FUNCTION_BLOCK Feedforward (* Composite Function Block Type *)
  (* Standard: 61499-2 *)
  (* Version 0.0, 2018-09-24, 4DIAC-IDE, 4DIAC-Consortium *)
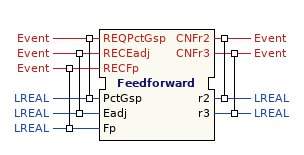
  EVENT_INPUT
    REQPctGsp WITH PctGsp;
    RECEadj WITH Eadj;
    RECFp WITH Fp;
  END_EVENT
  EVENT_OUTPUT
    CNFr2 WITH r2;
    CNFr3 WITH r3;
  END_EVENT
  VAR_INPUT
    PctGsp : LREAL;
    Eadj : LREAL;
    Fp : LREAL;
  END_VAR
  VAR_OUTPUT
    r2 : LREAL;
    r3 : LREAL;
  END_VAR
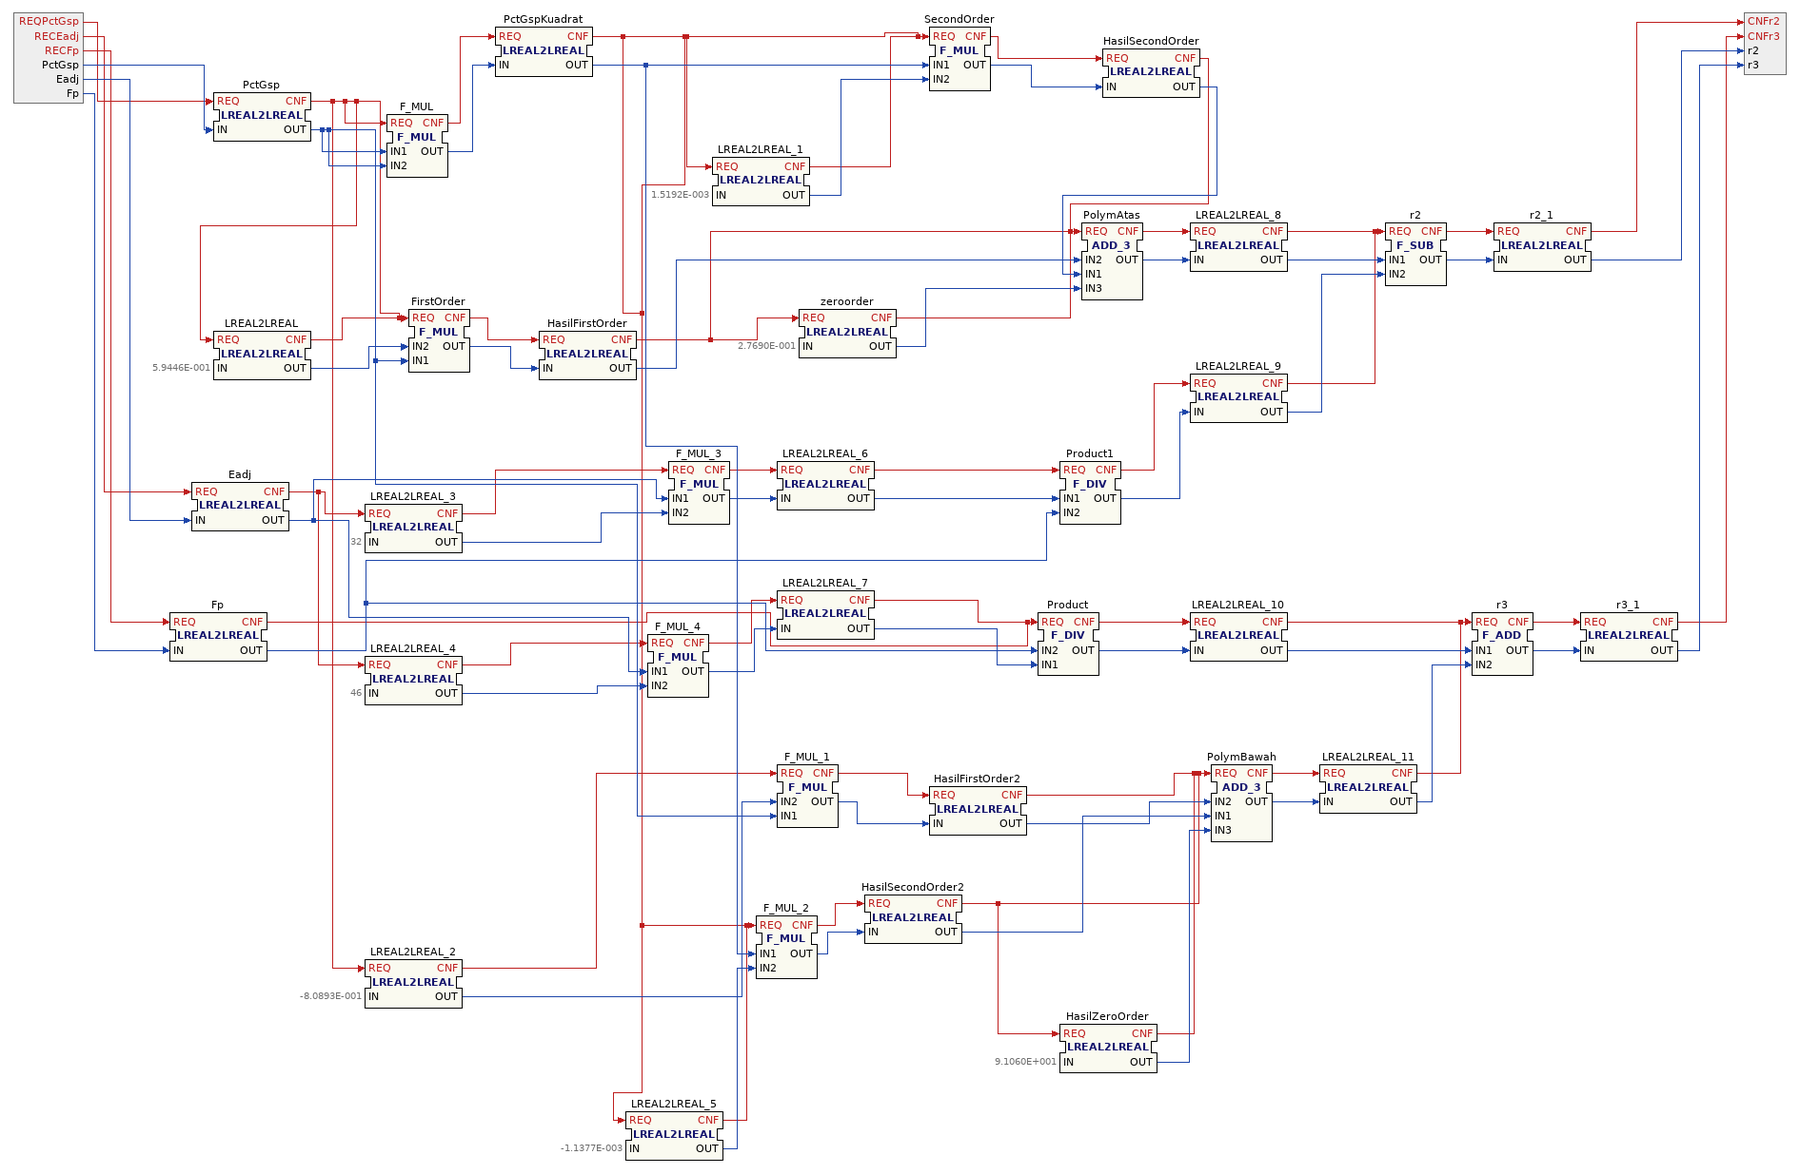
  FBS
    PctGsp : LREAL2LREAL;
    Eadj : LREAL2LREAL;
    Fp : LREAL2LREAL;
    F_MUL : F_MUL;
    PctGspKuadrat : LREAL2LREAL;
    LREAL2LREAL : LREAL2LREAL(IN := 5.9446E-001);
    LREAL2LREAL_1 : LREAL2LREAL(IN := 1.5192E-003);
    HasilFirstOrder : LREAL2LREAL;
    HasilSecondOrder : LREAL2LREAL;
    zeroorder : LREAL2LREAL(IN := 2.7690E-001);
    FirstOrder : F_MUL;
    PolymAtas : ADD_3;
    SecondOrder : F_MUL;
    PolymBawah : ADD_3;
    LREAL2LREAL_2 : LREAL2LREAL(IN := -8.0893E-001);
    F_MUL_1 : F_MUL;
    HasilFirstOrder2 : LREAL2LREAL;
    HasilSecondOrder2 : LREAL2LREAL;
    LREAL2LREAL_5 : LREAL2LREAL(IN := -1.1377E-003);
    F_MUL_2 : F_MUL;
    HasilZeroOrder : LREAL2LREAL(IN := 9.1060E+001);
    LREAL2LREAL_3 : LREAL2LREAL(IN := 32);
    LREAL2LREAL_4 : LREAL2LREAL(IN := 46);
    F_MUL_3 : F_MUL;
    F_MUL_4 : F_MUL;
    LREAL2LREAL_6 : LREAL2LREAL;
    LREAL2LREAL_7 : LREAL2LREAL;
    Product1 : F_DIV;
    Product : F_DIV;
    r2 : F_SUB;
    LREAL2LREAL_8 : LREAL2LREAL;
    LREAL2LREAL_9 : LREAL2LREAL;
    LREAL2LREAL_10 : LREAL2LREAL;
    r3 : F_ADD;
    LREAL2LREAL_11 : LREAL2LREAL;
    r2_1 : LREAL2LREAL;
    r3_1 : LREAL2LREAL;
  END_FBS
  EVENT_CONNECTIONS
    REQPctGsp TO PctGsp.REQ;
    RECEadj TO Eadj.REQ;
    RECFp TO Fp.REQ;
    PctGsp.CNF TO F_MUL.REQ;
    F_MUL.CNF TO PctGspKuadrat.REQ;
    PctGsp.CNF TO LREAL2LREAL.REQ;
    LREAL2LREAL.CNF TO FirstOrder.REQ;
    PctGsp.CNF TO FirstOrder.REQ;
    FirstOrder.CNF TO HasilFirstOrder.REQ;
    HasilFirstOrder.CNF TO PolymAtas.REQ;
    LREAL2LREAL_1.CNF TO SecondOrder.REQ;
    PctGspKuadrat.CNF TO SecondOrder.REQ;
    PctGspKuadrat.CNF TO LREAL2LREAL_1.REQ;
    SecondOrder.CNF TO HasilSecondOrder.REQ;
    HasilSecondOrder.CNF TO PolymAtas.REQ;
    zeroorder.CNF TO PolymAtas.REQ;
    HasilFirstOrder.CNF TO zeroorder.REQ;
    PctGsp.CNF TO LREAL2LREAL_2.REQ;
    LREAL2LREAL_2.CNF TO F_MUL_1.REQ;
    F_MUL_1.CNF TO HasilFirstOrder2.REQ;
    HasilFirstOrder2.CNF TO PolymBawah.REQ;
    HasilSecondOrder2.CNF TO PolymBawah.REQ;
    F_MUL_2.CNF TO HasilSecondOrder2.REQ;
    PctGspKuadrat.CNF TO F_MUL_2.REQ;
    LREAL2LREAL_5.CNF TO F_MUL_2.REQ;
    PctGspKuadrat.CNF TO LREAL2LREAL_5.REQ;
    HasilZeroOrder.CNF TO PolymBawah.REQ;
    HasilSecondOrder2.CNF TO HasilZeroOrder.REQ;
    Eadj.CNF TO LREAL2LREAL_4.REQ;
    Eadj.CNF TO LREAL2LREAL_3.REQ;
    LREAL2LREAL_4.CNF TO F_MUL_4.REQ;
    LREAL2LREAL_3.CNF TO F_MUL_3.REQ;
    F_MUL_3.CNF TO LREAL2LREAL_6.REQ;
    LREAL2LREAL_6.CNF TO Product1.REQ;
    F_MUL_4.CNF TO LREAL2LREAL_7.REQ;
    LREAL2LREAL_7.CNF TO Product.REQ;
    Fp.CNF TO Product.REQ;
    PolymAtas.CNF TO LREAL2LREAL_8.REQ;
    LREAL2LREAL_8.CNF TO r2.REQ;
    LREAL2LREAL_9.CNF TO r2.REQ;
    Product1.CNF TO LREAL2LREAL_9.REQ;
    Product.CNF TO LREAL2LREAL_10.REQ;
    LREAL2LREAL_10.CNF TO r3.REQ;
    PolymBawah.CNF TO LREAL2LREAL_11.REQ;
    LREAL2LREAL_11.CNF TO r3.REQ;
    r2_1.CNF TO CNFr2;
    r2.CNF TO r2_1.REQ;
    r3.CNF TO r3_1.REQ;
    r3_1.CNF TO CNFr3;
  END_CONNECTIONS
  DATA_CONNECTIONS
    Fp TO Fp.IN;
    PctGsp TO PctGsp.IN;
    PctGsp.OUT TO F_MUL.IN1;
    PctGsp.OUT TO F_MUL.IN2;
    F_MUL.OUT TO PctGspKuadrat.IN;
    LREAL2LREAL.OUT TO FirstOrder.IN2;
    PctGsp.OUT TO FirstOrder.IN1;
    FirstOrder.OUT TO HasilFirstOrder.IN;
    HasilFirstOrder.OUT TO PolymAtas.IN2;
    PctGspKuadrat.OUT TO SecondOrder.IN1;
    LREAL2LREAL_1.OUT TO SecondOrder.IN2;
    SecondOrder.OUT TO HasilSecondOrder.IN;
    HasilSecondOrder.OUT TO PolymAtas.IN1;
    zeroorder.OUT TO PolymAtas.IN3;
    LREAL2LREAL_2.OUT TO F_MUL_1.IN2;
    PctGsp.OUT TO F_MUL_1.IN1;
    F_MUL_1.OUT TO HasilFirstOrder2.IN;
    HasilFirstOrder2.OUT TO PolymBawah.IN2;
    HasilSecondOrder2.OUT TO PolymBawah.IN1;
    F_MUL_2.OUT TO HasilSecondOrder2.IN;
    PctGspKuadrat.OUT TO F_MUL_2.IN1;
    LREAL2LREAL_5.OUT TO F_MUL_2.IN2;
    HasilZeroOrder.OUT TO PolymBawah.IN3;
    Eadj TO Eadj.IN;
    Eadj.OUT TO F_MUL_3.IN1;
    Eadj.OUT TO F_MUL_4.IN1;
    LREAL2LREAL_3.OUT TO F_MUL_3.IN2;
    LREAL2LREAL_4.OUT TO F_MUL_4.IN2;
    F_MUL_3.OUT TO LREAL2LREAL_6.IN;
    LREAL2LREAL_6.OUT TO Product1.IN1;
    F_MUL_4.OUT TO LREAL2LREAL_7.IN;
    Fp.OUT TO Product.IN2;
    LREAL2LREAL_7.OUT TO Product.IN1;
    Fp.OUT TO Product1.IN2;
    PolymAtas.OUT TO LREAL2LREAL_8.IN;
    LREAL2LREAL_8.OUT TO r2.IN1;
    Product1.OUT TO LREAL2LREAL_9.IN;
    LREAL2LREAL_9.OUT TO r2.IN2;
    Product.OUT TO LREAL2LREAL_10.IN;
    LREAL2LREAL_10.OUT TO r3.IN1;
    PolymBawah.OUT TO LREAL2LREAL_11.IN;
    LREAL2LREAL_11.OUT TO r3.IN2;
    r2.OUT TO r2_1.IN;
    r2_1.OUT TO r2;
    r3.OUT TO r3_1.IN;
    r3_1.OUT TO r3;
  END_CONNECTIONS
END_FUNCTION_BLOCK
